// TIA Portal V20 export
FUNCTION_BLOCK "FB_ShredderSequencer"   // FB8, LAD
TITLE = Shredder Plant Sequencer
// Shredder plant sequencer (C-118-C-125): commands the shredder motor (via FB_MotorFwdRevSystem, wired at FC_ControlMain) and gates infeed/discharge conveyors and upstream enable, through a stepped cycle. Step legend (C-120): 0=Idle (stopped, waiting for a start condition) - 10=PreStart (siren warning before motion; arms the motor via MotorStartArm) - 20=DischargeStart (discharge conveyor starting, timed) - 30=ReverseRun (reverse commanded; the motor FB's own ReverseDelay entry pause elapses inside this step, then ReverseRunTimer counts ShredderReverseRunTime of CONFIRMED reverse feedback) - 40=WaitForwardRun (waiting for forward-run feedback) - 50=Running (normal production; infeed/upstream-enable timers and overcurrent detection are live) - 60=OvercurrentAbort (tripped - pause, then retry into ReverseRun, or stay out if too many reversals). Stop-all (REQ-012/013/062): StopCmd = stop button OR downstream lost OR control circuit unhealthy - aborts every step to Idle. Pusher handling is split (owner amendment 2026-07-16): stop button/unhealthy force pusher mode 0 (parks AND blocks jog), while any live stop reason - downstream loss included - raises PusherCycleInhibitCmd (no cycle launches or continues into a stopped plant, hand-jog stays available).
   VAR RETAIN
      IO { S7_SetPoint := 'True'} : "UDT_ShredderSequencerIO";   // Caller-visible interface (C-115) - FC_ControlMain writes CycleStart/CycleStop/feedback/tunables in, reads Run*/EnableUpstream/PreStartSounder/motor-command bits out. See the block header for the Step value legend.
   END_VAR
   VAR
      StopCmd : Bool;   // Stop-all: operator CycleStop, loss of DownstreamRunning (nowhere for shredded material to go), or loss of SystemHealthy (control circuit/E-stop - REQ-062: recovery must demand a fresh start press, so the sequence may not sit in a run step through an E-stop). Read by every step's own stop transition below and mirrored to the pusher as PusherCycleInhibitCmd.
      PusherModeForceOff : Bool;   // Named once (C-601): the hard pusher force - operator stop or circuit-unhealthy, plus the overcurrent-abort step. Forces PusherModeCmd to 0, which parks the pusher AND blocks jogging. Deliberately NOT the full StopCmd (owner amendment 2026-07-16): downstream absence must leave hand-jog available (REQ-040), so it reaches the pusher only as PusherCycleInhibitCmd.
      ReversalWindowTimeMS : DInt;
      PreStartSounderTimeMS : DInt;
      DischargeConveyorTimeoutMS : DInt;
      ShredderReverseRunTimeMS : DInt;
      InfeedRestartDelayMS : DInt;
      InfeedToUpstreamEnableDelayMS : DInt;
      OvercurrentSpinUpAllowanceMS : DInt;
      OvercurrentMediumDelayMS : DInt;
      OvercurrentHighDelayMS : DInt;
      ReversalRetryPauseTimeMS : DInt;
      ReversalWindowTimer { S7_SetPoint := 'True'} : TON_TIME;
      ReversalStepEdge : Bool;
      ReversalStepEdgeMem : Bool;
      ReversalCount : Int;   // Reversals since the window last re-armed (not per-cycle, unlike the pusher's own PressureTripCount) - ReversalWindowTimer restarts the window every time this is above zero, so ReversalCountThreshold reversals must occur within one ReversalWindowTime of each other to raise ShredderBlockedFault, not just ReversalCountThreshold times ever.
      PreStartTimer { S7_SetPoint := 'True'} : TON_TIME;
      DischargeStartTimer { S7_SetPoint := 'True'} : TON_TIME;
      ReverseRunTimer { S7_SetPoint := 'True'} : TON_TIME;
      InfeedRestartTimer { S7_SetPoint := 'True'} : TON_TIME;
      UpstreamEnableTimer { S7_SetPoint := 'True'} : TON_TIME;
      InfeedRunning : Bool;   // Latched once InfeedRestartTimer has timed out from the last hopper-clear - drives RunInfeedConv directly and (after a further UpstreamEnableTimer delay) EnableUpstream.
      SpinUpTimer { S7_SetPoint := 'True'} : TON_TIME;
      OvercurrentMediumTimer { S7_SetPoint := 'True'} : TON_TIME;
      OvercurrentHighTimer { S7_SetPoint := 'True'} : TON_TIME;
      OvercurrentTripped : Bool;   // KNOWN GAP, not wired to real current yet: both timers below are gated 'AND NOT AlwaysTrue' (permanently false placeholders) because DB_AnalogInput.ShredderMotorCurrent > DB_Settings.OvercurrentSetpointMedium/High is a genuine Real-vs-Real comparison this converter's synthesizer can't type correctly yet (hardcodes Int) - flagged and deferred rather than guessed at. This bit, and Step 50's own overcurrent-abort transition, are dead code until that's built.
      OvercurrentAbortPauseTimer { S7_SetPoint := 'True'} : TON_TIME;
   END_VAR
   VAR_TEMP
      "Time" : Real;
   END_VAR
BEGIN

REGION Network 1: Stop Command
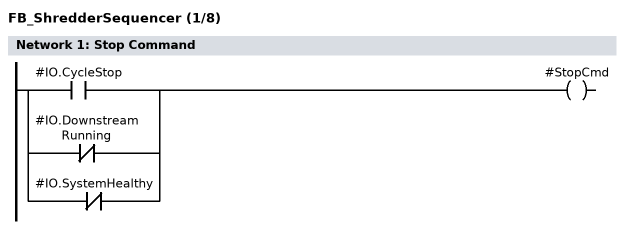
   RUNG wire#powerrail
      Contact( #IO.CycleStop )
      wire#w1
      Coil( #StopCmd )
   END_RUNG
   RUNG wire#powerrail
      I_Contact( #IO.DownstreamRunning )
   END_RUNG wire#w1
   RUNG wire#powerrail
      I_Contact( #IO.SystemHealthy )
   END_RUNG wire#w1
   // the same network as SCL:
   #StopCmd := #IO.CycleStop OR NOT #IO.DownstreamRunning OR NOT #IO.SystemHealthy;
END_REGION

REGION Network 2: HMI Time Conversions
   // HMI/DB_Settings times are Real seconds for operator legibility; every TON below needs its PT in DInt ms - one MUL+CONVERT pair per timer, matching the MotorDOL FTTime/EnableUPSTime idiom. Kept as one block up front rather than repeated at each timer, so the x1000 idiom is visibly consistent and only ever done once.
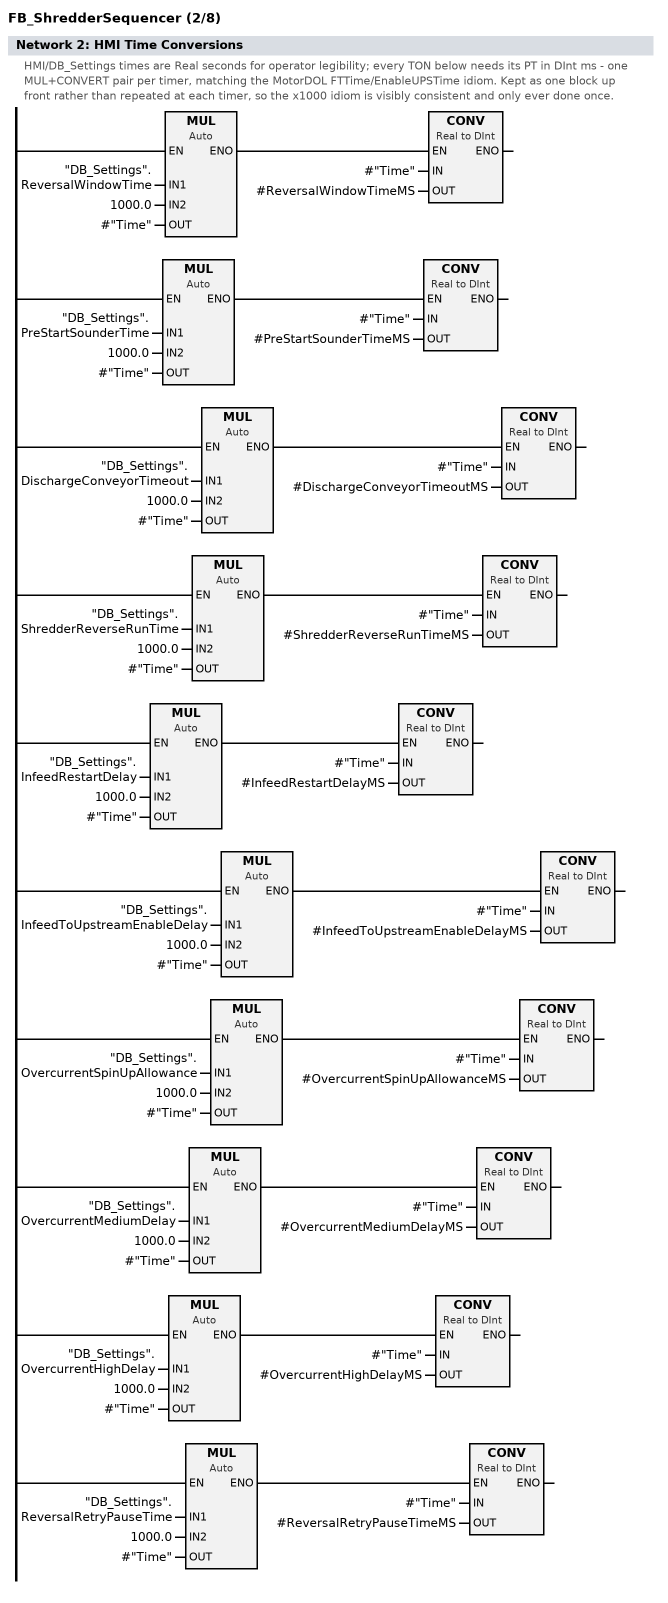
   RUNG wire#powerrail
      Mul(in1 := "DB_Settings".ReversalWindowTime, in2 := 1000.0, out := #"Time")
      { S7_Templates := "[SrcType := Real, DestType := DInt]" } Convert(in := #"Time", out := #ReversalWindowTimeMS)
   END_RUNG
   RUNG wire#powerrail
      Mul(in1 := "DB_Settings".PreStartSounderTime, in2 := 1000.0, out := #"Time")
      { S7_Templates := "[SrcType := Real, DestType := DInt]" } Convert(in := #"Time", out := #PreStartSounderTimeMS)
   END_RUNG
   RUNG wire#powerrail
      Mul(in1 := "DB_Settings".DischargeConveyorTimeout, in2 := 1000.0, out := #"Time")
      { S7_Templates := "[SrcType := Real, DestType := DInt]" } Convert(in := #"Time", out := #DischargeConveyorTimeoutMS)
   END_RUNG
   RUNG wire#powerrail
      Mul(in1 := "DB_Settings".ShredderReverseRunTime, in2 := 1000.0, out := #"Time")
      { S7_Templates := "[SrcType := Real, DestType := DInt]" } Convert(in := #"Time", out := #ShredderReverseRunTimeMS)
   END_RUNG
   RUNG wire#powerrail
      Mul(in1 := "DB_Settings".InfeedRestartDelay, in2 := 1000.0, out := #"Time")
      { S7_Templates := "[SrcType := Real, DestType := DInt]" } Convert(in := #"Time", out := #InfeedRestartDelayMS)
   END_RUNG
   RUNG wire#powerrail
      Mul(in1 := "DB_Settings".InfeedToUpstreamEnableDelay, in2 := 1000.0, out := #"Time")
      { S7_Templates := "[SrcType := Real, DestType := DInt]" } Convert(in := #"Time", out := #InfeedToUpstreamEnableDelayMS)
   END_RUNG
   RUNG wire#powerrail
      Mul(in1 := "DB_Settings".OvercurrentSpinUpAllowance, in2 := 1000.0, out := #"Time")
      { S7_Templates := "[SrcType := Real, DestType := DInt]" } Convert(in := #"Time", out := #OvercurrentSpinUpAllowanceMS)
   END_RUNG
   RUNG wire#powerrail
      Mul(in1 := "DB_Settings".OvercurrentMediumDelay, in2 := 1000.0, out := #"Time")
      { S7_Templates := "[SrcType := Real, DestType := DInt]" } Convert(in := #"Time", out := #OvercurrentMediumDelayMS)
   END_RUNG
   RUNG wire#powerrail
      Mul(in1 := "DB_Settings".OvercurrentHighDelay, in2 := 1000.0, out := #"Time")
      { S7_Templates := "[SrcType := Real, DestType := DInt]" } Convert(in := #"Time", out := #OvercurrentHighDelayMS)
   END_RUNG
   RUNG wire#powerrail
      Mul(in1 := "DB_Settings".ReversalRetryPauseTime, in2 := 1000.0, out := #"Time")
      { S7_Templates := "[SrcType := Real, DestType := DInt]" } Convert(in := #"Time", out := #ReversalRetryPauseTimeMS)
   END_RUNG
   // the same network as SCL:
   <??.?> := "DB_Settings".ReversalWindowTime * 1000.0 * #"Time";
   <??.?> := REAL_TO_DINT(#"Time");
   <??.?> := "DB_Settings".PreStartSounderTime * 1000.0 * #"Time";
   <??.?> := REAL_TO_DINT(#"Time");
   <??.?> := "DB_Settings".DischargeConveyorTimeout * 1000.0 * #"Time";
   <??.?> := REAL_TO_DINT(#"Time");
   <??.?> := "DB_Settings".ShredderReverseRunTime * 1000.0 * #"Time";
   <??.?> := REAL_TO_DINT(#"Time");
   <??.?> := "DB_Settings".InfeedRestartDelay * 1000.0 * #"Time";
   <??.?> := REAL_TO_DINT(#"Time");
   <??.?> := "DB_Settings".InfeedToUpstreamEnableDelay * 1000.0 * #"Time";
   <??.?> := REAL_TO_DINT(#"Time");
   <??.?> := "DB_Settings".OvercurrentSpinUpAllowance * 1000.0 * #"Time";
   <??.?> := REAL_TO_DINT(#"Time");
   <??.?> := "DB_Settings".OvercurrentMediumDelay * 1000.0 * #"Time";
   <??.?> := REAL_TO_DINT(#"Time");
   <??.?> := "DB_Settings".OvercurrentHighDelay * 1000.0 * #"Time";
   <??.?> := REAL_TO_DINT(#"Time");
   <??.?> := "DB_Settings".ReversalRetryPauseTime * 1000.0 * #"Time";
   <??.?> := REAL_TO_DINT(#"Time");
END_REGION

REGION Network 3: Reversal Re-Arm Window Timer
   // Retriggerable on-delay built from TON+edge (C-406/C-404 - no TONR/TOF exists to do this natively). IN drops false the instant a NEW reversal is detected - Step transitioning into 60, tested against ReversalStepEdgeMem's own previous-scan value (correct read-before-write ordering: this network reads the memory bit before Network 4 updates it later the same scan, so no cross-network staleness) - which resets ET/Q to 0 that scan; the timer then re-arms and must run a full ReversalWindowTime with no further reversal before Q goes true. Fixed 2026-07-17 (owner ruling, B-5/REQ-028): the prior rung read IN := ReversalCount > 0 alone, a level condition that only ever ran once from the first reversal - a fixed window, not the re-arming one this network's own title always claimed (C-608).
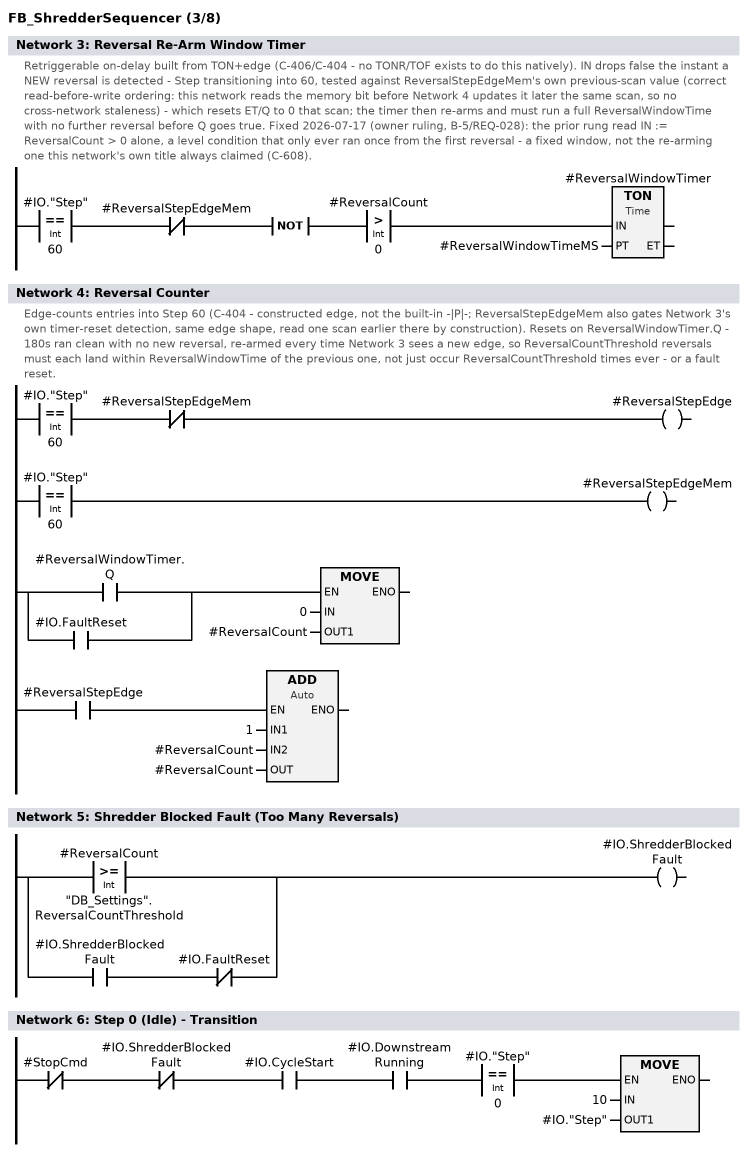
   RUNG wire#powerrail
      { S7_Templates := "SrcType := Int" } EQ_Contact(in1 := #IO."Step", in2 := 60)
      I_Contact( #ReversalStepEdgeMem )
      Not()
      { S7_Templates := "SrcType := Int" } GT_Contact(in1 := #ReversalCount, in2 := 0)
      { S7_Templates := "time_type := Time" } #ReversalWindowTimer.TON(pt := #ReversalWindowTimeMS, et =>)
   END_RUNG
   // the same network as SCL:
   #ReversalWindowTimer(IN := NOT ((#IO."Step" = 60) AND NOT #ReversalStepEdgeMem) AND (#ReversalCount > 0),   // TON
                        PT := #ReversalWindowTimeMS);
END_REGION

REGION Network 4: Reversal Counter
   // Edge-counts entries into Step 60 (C-404 - constructed edge, not the built-in -|P|-; ReversalStepEdgeMem also gates Network 3's own timer-reset detection, same edge shape, read one scan earlier there by construction). Resets on ReversalWindowTimer.Q - 180s ran clean with no new reversal, re-armed every time Network 3 sees a new edge, so ReversalCountThreshold reversals must each land within ReversalWindowTime of the previous one, not just occur ReversalCountThreshold times ever - or a fault reset.
   RUNG wire#powerrail
      { S7_Templates := "SrcType := Int" } EQ_Contact(in1 := #IO."Step", in2 := 60)
      I_Contact( #ReversalStepEdgeMem )
      Coil( #ReversalStepEdge )
   END_RUNG
   RUNG wire#powerrail
      { S7_Templates := "SrcType := Int" } EQ_Contact(in1 := #IO."Step", in2 := 60)
      Coil( #ReversalStepEdgeMem )
   END_RUNG
   RUNG wire#powerrail
      Contact( #ReversalWindowTimer.Q )
      wire#w1
      Move(in := 0, out1 := #ReversalCount)
   END_RUNG
   RUNG wire#powerrail
      Contact( #IO.FaultReset )
   END_RUNG wire#w1
   RUNG wire#powerrail
      Contact( #ReversalStepEdge )
      Add(in1 := 1, in2 := #ReversalCount, out := #ReversalCount)
   END_RUNG
   // the same network as SCL:
   #ReversalStepEdge := (#IO."Step" = 60) AND NOT #ReversalStepEdgeMem;
   #ReversalStepEdgeMem := #IO."Step" = 60;
   IF #ReversalWindowTimer.Q OR #IO.FaultReset THEN <??.?> := 0; END_IF;
   IF #ReversalStepEdge THEN <??.?> := 1 + #ReversalCount + #ReversalCount; END_IF;
END_REGION

REGION Network 5: Shredder Blocked Fault (Too Many Reversals)
   RUNG wire#powerrail
      { S7_Templates := "SrcType := Int" } GE_Contact(in1 := #ReversalCount, in2 := "DB_Settings".ReversalCountThreshold)
      wire#w1
      Coil( #IO.ShredderBlockedFault )
   END_RUNG
   RUNG wire#powerrail
      Contact( #IO.ShredderBlockedFault )
      I_Contact( #IO.FaultReset )
   END_RUNG wire#w1
   // the same network as SCL:
   #IO.ShredderBlockedFault := (#ReversalCount >= "DB_Settings".ReversalCountThreshold) OR (#IO.ShredderBlockedFault AND NOT #IO.FaultReset);
END_REGION

REGION Network 6: Step 0 (Idle) - Transition
   RUNG wire#powerrail
      I_Contact( #StopCmd )
      I_Contact( #IO.ShredderBlockedFault )
      Contact( #IO.CycleStart )
      Contact( #IO.DownstreamRunning )
      { S7_Templates := "SrcType := Int" } EQ_Contact(in1 := #IO."Step", in2 := 0)
      Move(in := 10, out1 := #IO."Step")
   END_RUNG
   // the same network as SCL:
   IF NOT #StopCmd AND NOT #IO.ShredderBlockedFault AND #IO.CycleStart AND #IO.DownstreamRunning AND (#IO."Step" = 0) THEN
       <??.?> := 10;
   END_IF;
END_REGION

REGION Network 7: Step 10 (PreStart) - Timer And Transitions
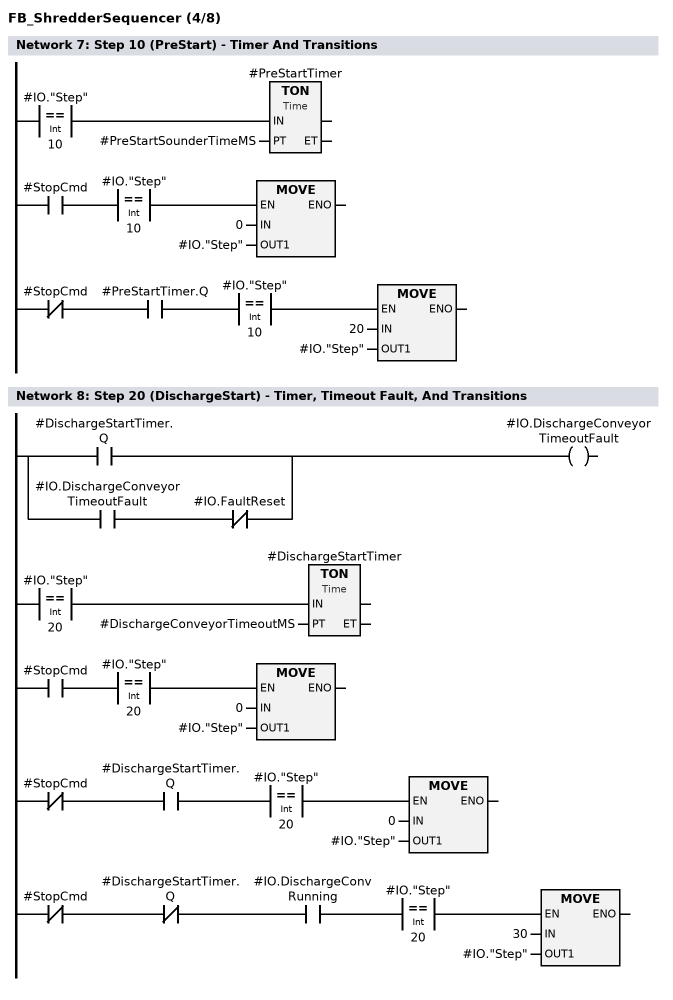
   RUNG wire#powerrail
      { S7_Templates := "SrcType := Int" } EQ_Contact(in1 := #IO."Step", in2 := 10)
      { S7_Templates := "time_type := Time" } #PreStartTimer.TON(pt := #PreStartSounderTimeMS, et =>)
   END_RUNG
   RUNG wire#powerrail
      Contact( #StopCmd )
      { S7_Templates := "SrcType := Int" } EQ_Contact(in1 := #IO."Step", in2 := 10)
      Move(in := 0, out1 := #IO."Step")
   END_RUNG
   RUNG wire#powerrail
      I_Contact( #StopCmd )
      Contact( #PreStartTimer.Q )
      { S7_Templates := "SrcType := Int" } EQ_Contact(in1 := #IO."Step", in2 := 10)
      Move(in := 20, out1 := #IO."Step")
   END_RUNG
   // the same network as SCL:
   #PreStartTimer(IN := #IO."Step" = 10, PT := #PreStartSounderTimeMS);   // TON
   IF #StopCmd AND (#IO."Step" = 10) THEN <??.?> := 0; END_IF;
   IF NOT #StopCmd AND #PreStartTimer.Q AND (#IO."Step" = 10) THEN <??.?> := 20; END_IF;
END_REGION

REGION Network 8: Step 20 (DischargeStart) - Timer, Timeout Fault, And Transitions
   RUNG wire#powerrail
      Contact( #DischargeStartTimer.Q )
      wire#w1
      Coil( #IO.DischargeConveyorTimeoutFault )
   END_RUNG
   RUNG wire#powerrail
      Contact( #IO.DischargeConveyorTimeoutFault )
      I_Contact( #IO.FaultReset )
   END_RUNG wire#w1
   RUNG wire#powerrail
      { S7_Templates := "SrcType := Int" } EQ_Contact(in1 := #IO."Step", in2 := 20)
      { S7_Templates := "time_type := Time" } #DischargeStartTimer.TON(pt := #DischargeConveyorTimeoutMS, et =>)
   END_RUNG
   RUNG wire#powerrail
      Contact( #StopCmd )
      { S7_Templates := "SrcType := Int" } EQ_Contact(in1 := #IO."Step", in2 := 20)
      Move(in := 0, out1 := #IO."Step")
   END_RUNG
   RUNG wire#powerrail
      I_Contact( #StopCmd )
      Contact( #DischargeStartTimer.Q )
      { S7_Templates := "SrcType := Int" } EQ_Contact(in1 := #IO."Step", in2 := 20)
      Move(in := 0, out1 := #IO."Step")
   END_RUNG
   RUNG wire#powerrail
      I_Contact( #StopCmd )
      I_Contact( #DischargeStartTimer.Q )
      Contact( #IO.DischargeConvRunning )
      { S7_Templates := "SrcType := Int" } EQ_Contact(in1 := #IO."Step", in2 := 20)
      Move(in := 30, out1 := #IO."Step")
   END_RUNG
   // the same network as SCL:
   #IO.DischargeConveyorTimeoutFault := #DischargeStartTimer.Q OR (#IO.DischargeConveyorTimeoutFault AND NOT #IO.FaultReset);
   #DischargeStartTimer(IN := #IO."Step" = 20, PT := #DischargeConveyorTimeoutMS);   // TON
   IF #StopCmd AND (#IO."Step" = 20) THEN <??.?> := 0; END_IF;
   IF NOT #StopCmd AND #DischargeStartTimer.Q AND (#IO."Step" = 20) THEN <??.?> := 0; END_IF;
   IF NOT #StopCmd AND NOT #DischargeStartTimer.Q AND #IO.DischargeConvRunning AND (#IO."Step" = 20) THEN
       <??.?> := 30;
   END_IF;
END_REGION

REGION Network 9: Step 30 (ReverseRun) - Timer And Transitions
   // ReverseRunTimer counts only while reverse is CONFIRMED running (ShredderRunRevFB), so the spec's 6 s (REQ-005) buys 6 s of actual rotation - the motor FB's 8 s ReverseDelay entry pause no longer eats the window, and a feedback dropout restarts the count. The commanded-but-no-feedback dwell is deliberately NOT re-timed here (C-409, one interval one place; step 40 already relies on the same mechanism): the motor FB's own fail-to-run window (FTTime, after its ReverseIgnoreFT masking) latches FTR, and the MotorFaultActive exit below aborts the step - bounded dwell, latched fault, C-122's substance without a duplicate timer.
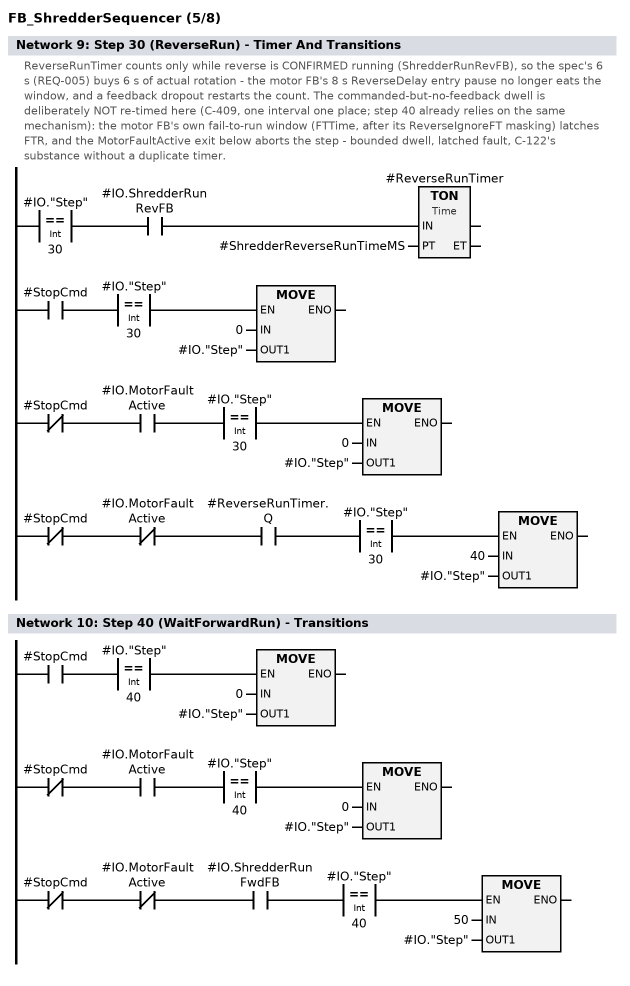
   RUNG wire#powerrail
      { S7_Templates := "SrcType := Int" } EQ_Contact(in1 := #IO."Step", in2 := 30)
      Contact( #IO.ShredderRunRevFB )
      { S7_Templates := "time_type := Time" } #ReverseRunTimer.TON(pt := #ShredderReverseRunTimeMS, et =>)
   END_RUNG
   RUNG wire#powerrail
      Contact( #StopCmd )
      { S7_Templates := "SrcType := Int" } EQ_Contact(in1 := #IO."Step", in2 := 30)
      Move(in := 0, out1 := #IO."Step")
   END_RUNG
   RUNG wire#powerrail
      I_Contact( #StopCmd )
      Contact( #IO.MotorFaultActive )
      { S7_Templates := "SrcType := Int" } EQ_Contact(in1 := #IO."Step", in2 := 30)
      Move(in := 0, out1 := #IO."Step")
   END_RUNG
   RUNG wire#powerrail
      I_Contact( #StopCmd )
      I_Contact( #IO.MotorFaultActive )
      Contact( #ReverseRunTimer.Q )
      { S7_Templates := "SrcType := Int" } EQ_Contact(in1 := #IO."Step", in2 := 30)
      Move(in := 40, out1 := #IO."Step")
   END_RUNG
   // the same network as SCL:
   #ReverseRunTimer(IN := (#IO."Step" = 30) AND #IO.ShredderRunRevFB, PT := #ShredderReverseRunTimeMS);   // TON
   IF #StopCmd AND (#IO."Step" = 30) THEN <??.?> := 0; END_IF;
   IF NOT #StopCmd AND #IO.MotorFaultActive AND (#IO."Step" = 30) THEN <??.?> := 0; END_IF;
   IF NOT #StopCmd AND NOT #IO.MotorFaultActive AND #ReverseRunTimer.Q AND (#IO."Step" = 30) THEN
       <??.?> := 40;
   END_IF;
END_REGION

REGION Network 10: Step 40 (WaitForwardRun) - Transitions
   RUNG wire#powerrail
      Contact( #StopCmd )
      { S7_Templates := "SrcType := Int" } EQ_Contact(in1 := #IO."Step", in2 := 40)
      Move(in := 0, out1 := #IO."Step")
   END_RUNG
   RUNG wire#powerrail
      I_Contact( #StopCmd )
      Contact( #IO.MotorFaultActive )
      { S7_Templates := "SrcType := Int" } EQ_Contact(in1 := #IO."Step", in2 := 40)
      Move(in := 0, out1 := #IO."Step")
   END_RUNG
   RUNG wire#powerrail
      I_Contact( #StopCmd )
      I_Contact( #IO.MotorFaultActive )
      Contact( #IO.ShredderRunFwdFB )
      { S7_Templates := "SrcType := Int" } EQ_Contact(in1 := #IO."Step", in2 := 40)
      Move(in := 50, out1 := #IO."Step")
   END_RUNG
   // the same network as SCL:
   IF #StopCmd AND (#IO."Step" = 40) THEN <??.?> := 0; END_IF;
   IF NOT #StopCmd AND #IO.MotorFaultActive AND (#IO."Step" = 40) THEN <??.?> := 0; END_IF;
   IF NOT #StopCmd AND NOT #IO.MotorFaultActive AND #IO.ShredderRunFwdFB AND (#IO."Step" = 40) THEN
       <??.?> := 50;
   END_IF;
END_REGION

REGION Network 11: Step 50 (Running) - Infeed Restart, Upstream Enable, And Outputs
   // UpstreamEnableTimer's own IN reads InfeedRunning one scan behind this network's own InfeedRunning update below (it's kind-ordered before the coil that writes it) - harmless for a multi-second delay, and matches this design's original timing exactly. EnableUpstream lives here, next to its own timer, rather than in the general Output Commands network - this is the output the MotorFwdRevSystem CALL-site correction was specifically about: it must only ever come from Step=50 dwell time, never from motor-running telemetry.
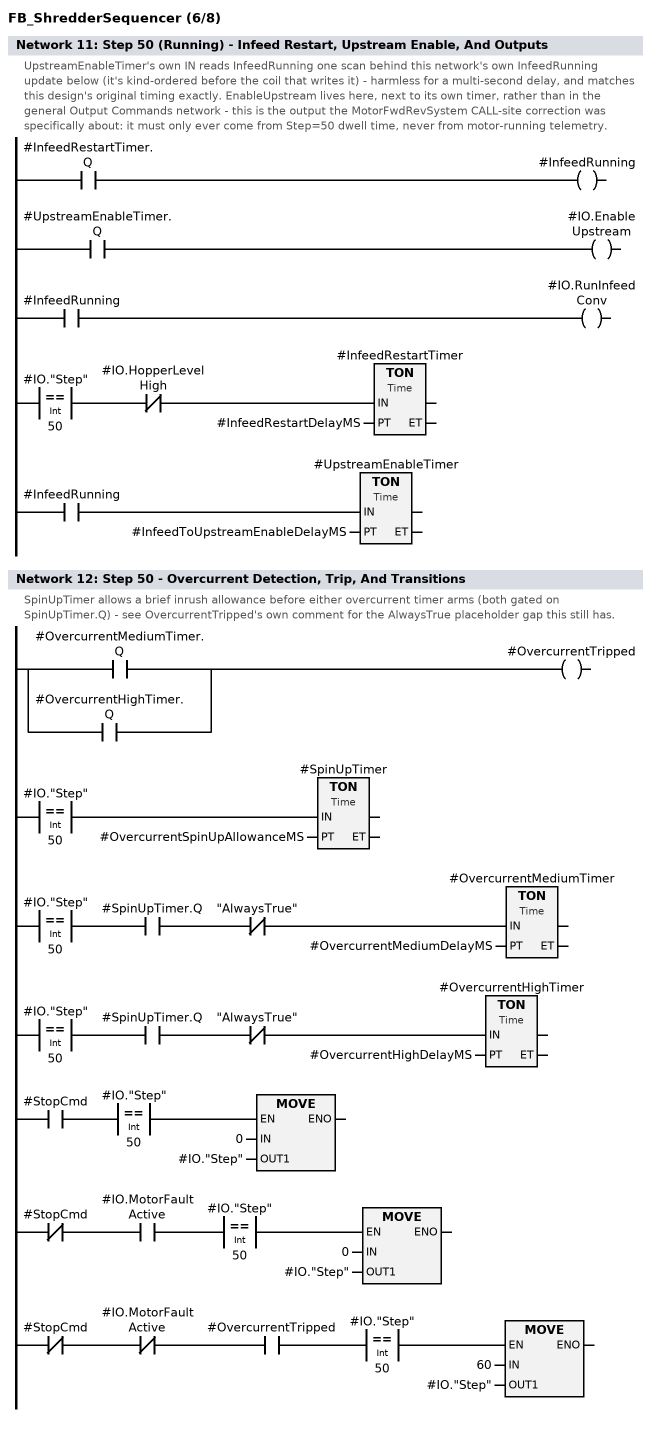
   RUNG wire#powerrail
      Contact( #InfeedRestartTimer.Q )
      Coil( #InfeedRunning )
   END_RUNG
   RUNG wire#powerrail
      Contact( #UpstreamEnableTimer.Q )
      Coil( #IO.EnableUpstream )
   END_RUNG
   RUNG wire#powerrail
      Contact( #InfeedRunning )
      Coil( #IO.RunInfeedConv )
   END_RUNG
   RUNG wire#powerrail
      { S7_Templates := "SrcType := Int" } EQ_Contact(in1 := #IO."Step", in2 := 50)
      I_Contact( #IO.HopperLevelHigh )
      { S7_Templates := "time_type := Time" } #InfeedRestartTimer.TON(pt := #InfeedRestartDelayMS, et =>)
   END_RUNG
   RUNG wire#powerrail
      Contact( #InfeedRunning )
      { S7_Templates := "time_type := Time" } #UpstreamEnableTimer.TON(pt := #InfeedToUpstreamEnableDelayMS, et =>)
   END_RUNG
   // the same network as SCL:
   #InfeedRunning := #InfeedRestartTimer.Q;
   #IO.EnableUpstream := #UpstreamEnableTimer.Q;
   #IO.RunInfeedConv := #InfeedRunning;
   #InfeedRestartTimer(IN := (#IO."Step" = 50) AND NOT #IO.HopperLevelHigh, PT := #InfeedRestartDelayMS);   // TON
   #UpstreamEnableTimer(IN := #InfeedRunning, PT := #InfeedToUpstreamEnableDelayMS);   // TON
END_REGION

REGION Network 12: Step 50 - Overcurrent Detection, Trip, And Transitions
   // SpinUpTimer allows a brief inrush allowance before either overcurrent timer arms (both gated on SpinUpTimer.Q) - see OvercurrentTripped's own comment for the AlwaysTrue placeholder gap this still has.
   RUNG wire#powerrail
      Contact( #OvercurrentMediumTimer.Q )
      wire#w1
      Coil( #OvercurrentTripped )
   END_RUNG
   RUNG wire#powerrail
      Contact( #OvercurrentHighTimer.Q )
   END_RUNG wire#w1
   RUNG wire#powerrail
      { S7_Templates := "SrcType := Int" } EQ_Contact(in1 := #IO."Step", in2 := 50)
      { S7_Templates := "time_type := Time" } #SpinUpTimer.TON(pt := #OvercurrentSpinUpAllowanceMS, et =>)
   END_RUNG
   RUNG wire#powerrail
      { S7_Templates := "SrcType := Int" } EQ_Contact(in1 := #IO."Step", in2 := 50)
      Contact( #SpinUpTimer.Q )
      I_Contact( "AlwaysTrue" )
      { S7_Templates := "time_type := Time" } #OvercurrentMediumTimer.TON(pt := #OvercurrentMediumDelayMS, et =>)
   END_RUNG
   RUNG wire#powerrail
      { S7_Templates := "SrcType := Int" } EQ_Contact(in1 := #IO."Step", in2 := 50)
      Contact( #SpinUpTimer.Q )
      I_Contact( "AlwaysTrue" )
      { S7_Templates := "time_type := Time" } #OvercurrentHighTimer.TON(pt := #OvercurrentHighDelayMS, et =>)
   END_RUNG
   RUNG wire#powerrail
      Contact( #StopCmd )
      { S7_Templates := "SrcType := Int" } EQ_Contact(in1 := #IO."Step", in2 := 50)
      Move(in := 0, out1 := #IO."Step")
   END_RUNG
   RUNG wire#powerrail
      I_Contact( #StopCmd )
      Contact( #IO.MotorFaultActive )
      { S7_Templates := "SrcType := Int" } EQ_Contact(in1 := #IO."Step", in2 := 50)
      Move(in := 0, out1 := #IO."Step")
   END_RUNG
   RUNG wire#powerrail
      I_Contact( #StopCmd )
      I_Contact( #IO.MotorFaultActive )
      Contact( #OvercurrentTripped )
      { S7_Templates := "SrcType := Int" } EQ_Contact(in1 := #IO."Step", in2 := 50)
      Move(in := 60, out1 := #IO."Step")
   END_RUNG
   // the same network as SCL:
   #OvercurrentTripped := #OvercurrentMediumTimer.Q OR #OvercurrentHighTimer.Q;
   #SpinUpTimer(IN := #IO."Step" = 50, PT := #OvercurrentSpinUpAllowanceMS);   // TON
   #OvercurrentMediumTimer(IN := (#IO."Step" = 50) AND #SpinUpTimer.Q AND NOT "AlwaysTrue",   // TON
                           PT := #OvercurrentMediumDelayMS);
   #OvercurrentHighTimer(IN := (#IO."Step" = 50) AND #SpinUpTimer.Q AND NOT "AlwaysTrue",   // TON
                         PT := #OvercurrentHighDelayMS);
   IF #StopCmd AND (#IO."Step" = 50) THEN <??.?> := 0; END_IF;
   IF NOT #StopCmd AND #IO.MotorFaultActive AND (#IO."Step" = 50) THEN <??.?> := 0; END_IF;
   IF NOT #StopCmd AND NOT #IO.MotorFaultActive AND #OvercurrentTripped AND (#IO."Step" = 50) THEN
       <??.?> := 60;
   END_IF;
END_REGION

REGION Network 13: Step 60 (OvercurrentAbort) - Timer And Transitions
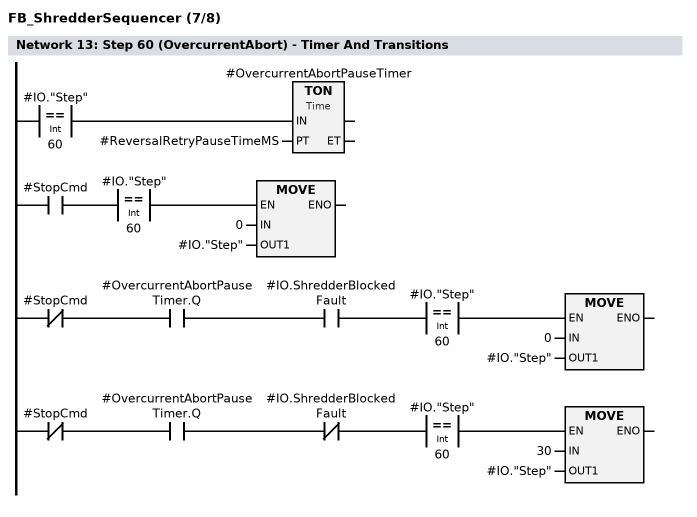
   RUNG wire#powerrail
      { S7_Templates := "SrcType := Int" } EQ_Contact(in1 := #IO."Step", in2 := 60)
      { S7_Templates := "time_type := Time" } #OvercurrentAbortPauseTimer.TON(pt := #ReversalRetryPauseTimeMS, et =>)
   END_RUNG
   RUNG wire#powerrail
      Contact( #StopCmd )
      { S7_Templates := "SrcType := Int" } EQ_Contact(in1 := #IO."Step", in2 := 60)
      Move(in := 0, out1 := #IO."Step")
   END_RUNG
   RUNG wire#powerrail
      I_Contact( #StopCmd )
      Contact( #OvercurrentAbortPauseTimer.Q )
      Contact( #IO.ShredderBlockedFault )
      { S7_Templates := "SrcType := Int" } EQ_Contact(in1 := #IO."Step", in2 := 60)
      Move(in := 0, out1 := #IO."Step")
   END_RUNG
   RUNG wire#powerrail
      I_Contact( #StopCmd )
      Contact( #OvercurrentAbortPauseTimer.Q )
      I_Contact( #IO.ShredderBlockedFault )
      { S7_Templates := "SrcType := Int" } EQ_Contact(in1 := #IO."Step", in2 := 60)
      Move(in := 30, out1 := #IO."Step")
   END_RUNG
   // the same network as SCL:
   #OvercurrentAbortPauseTimer(IN := #IO."Step" = 60, PT := #ReversalRetryPauseTimeMS);   // TON
   IF #StopCmd AND (#IO."Step" = 60) THEN <??.?> := 0; END_IF;
   IF NOT #StopCmd AND #OvercurrentAbortPauseTimer.Q AND #IO.ShredderBlockedFault AND (#IO."Step" = 60) THEN
       <??.?> := 0;
   END_IF;
   IF NOT #StopCmd AND #OvercurrentAbortPauseTimer.Q AND NOT #IO.ShredderBlockedFault AND (#IO."Step" = 60) THEN
       <??.?> := 30;
   END_IF;
END_REGION

REGION Network 14: Motor And Pusher Mode Commands
   // MotorStartArm asserts only through PreStart: one operator start press = one motor arming (FC_ControlMain hands it to the motor FB's self-clearing RecentStart - REQ-062). PusherParkCmd holds through the machine-start steps 20-40 (range intent, C-603: any step inserted inside the start ramp still wants the pusher home) - long enough for the pusher's warned repark to fire even when the discharge confirm is quick (REQ-045); from Running onward the pusher's own cycle-entry repark takes over. Pusher stop handling is two-tier (REQ-012/013 + owner amendment 2026-07-16): PusherModeForceOff (stop button/unhealthy/step-60, mirroring the step-60 overcurrent force) drives mode 0 - parks the pusher and blocks jog - while PusherCycleInhibitCmd mirrors the full StopCmd so downstream loss still stops cycle behavior without taking hand-jog away (REQ-040).
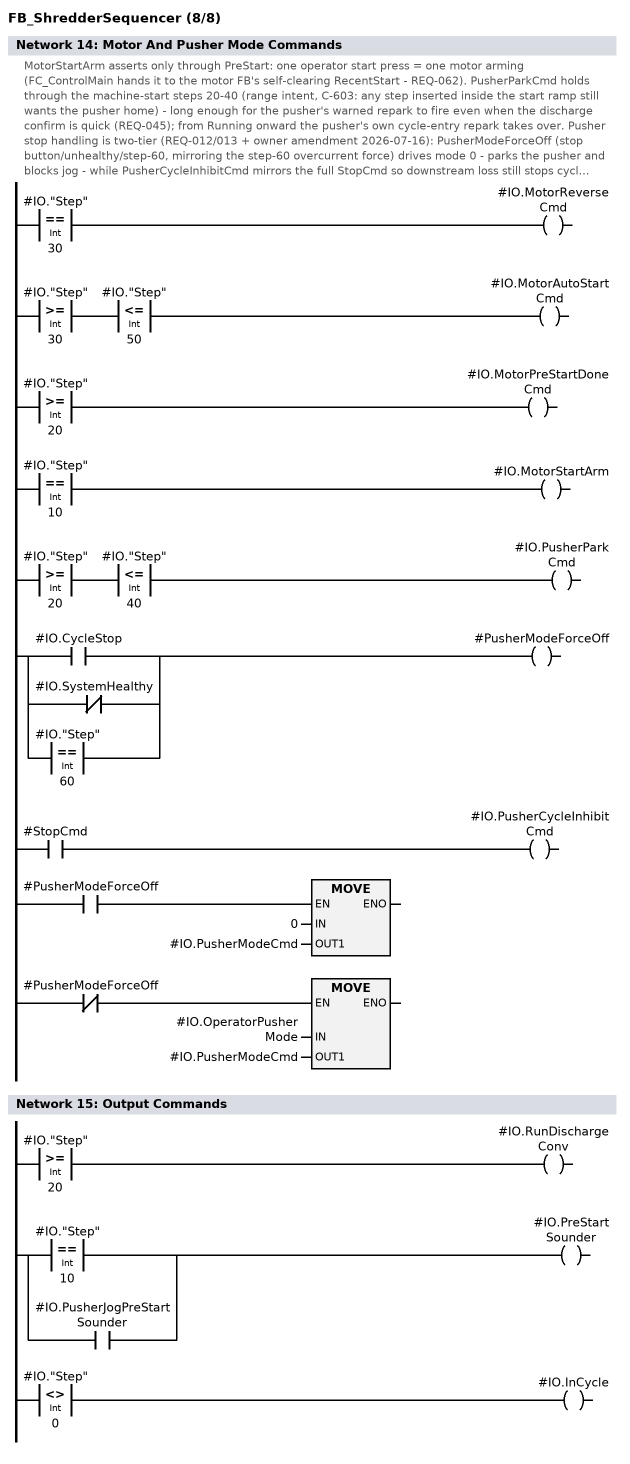
   RUNG wire#powerrail
      { S7_Templates := "SrcType := Int" } EQ_Contact(in1 := #IO."Step", in2 := 30)
      Coil( #IO.MotorReverseCmd )
   END_RUNG
   RUNG wire#powerrail
      { S7_Templates := "SrcType := Int" } GE_Contact(in1 := #IO."Step", in2 := 30)
      { S7_Templates := "SrcType := Int" } LE_Contact(in1 := #IO."Step", in2 := 50)
      Coil( #IO.MotorAutoStartCmd )
   END_RUNG
   RUNG wire#powerrail
      { S7_Templates := "SrcType := Int" } GE_Contact(in1 := #IO."Step", in2 := 20)
      Coil( #IO.MotorPreStartDoneCmd )
   END_RUNG
   RUNG wire#powerrail
      { S7_Templates := "SrcType := Int" } EQ_Contact(in1 := #IO."Step", in2 := 10)
      Coil( #IO.MotorStartArm )
   END_RUNG
   RUNG wire#powerrail
      { S7_Templates := "SrcType := Int" } GE_Contact(in1 := #IO."Step", in2 := 20)
      { S7_Templates := "SrcType := Int" } LE_Contact(in1 := #IO."Step", in2 := 40)
      Coil( #IO.PusherParkCmd )
   END_RUNG
   RUNG wire#powerrail
      Contact( #IO.CycleStop )
      wire#w1
      Coil( #PusherModeForceOff )
   END_RUNG
   RUNG wire#powerrail
      I_Contact( #IO.SystemHealthy )
   END_RUNG wire#w1
   RUNG wire#powerrail
      { S7_Templates := "SrcType := Int" } EQ_Contact(in1 := #IO."Step", in2 := 60)
   END_RUNG wire#w1
   RUNG wire#powerrail
      Contact( #StopCmd )
      Coil( #IO.PusherCycleInhibitCmd )
   END_RUNG
   RUNG wire#powerrail
      Contact( #PusherModeForceOff )
      Move(in := 0, out1 := #IO.PusherModeCmd)
   END_RUNG
   RUNG wire#powerrail
      I_Contact( #PusherModeForceOff )
      Move(in := #IO.OperatorPusherMode, out1 := #IO.PusherModeCmd)
   END_RUNG
   // the same network as SCL:
   #IO.MotorReverseCmd := #IO."Step" = 30;
   #IO.MotorAutoStartCmd := (#IO."Step" >= 30) AND (#IO."Step" <= 50);
   #IO.MotorPreStartDoneCmd := #IO."Step" >= 20;
   #IO.MotorStartArm := #IO."Step" = 10;
   #IO.PusherParkCmd := (#IO."Step" >= 20) AND (#IO."Step" <= 40);
   #PusherModeForceOff := #IO.CycleStop OR NOT #IO.SystemHealthy OR (#IO."Step" = 60);
   #IO.PusherCycleInhibitCmd := #StopCmd;
   IF #PusherModeForceOff THEN <??.?> := 0; END_IF;
   IF NOT #PusherModeForceOff THEN <??.?> := #IO.OperatorPusherMode; END_IF;
END_REGION

REGION Network 15: Output Commands
   RUNG wire#powerrail
      { S7_Templates := "SrcType := Int" } GE_Contact(in1 := #IO."Step", in2 := 20)
      Coil( #IO.RunDischargeConv )
   END_RUNG
   RUNG wire#powerrail
      { S7_Templates := "SrcType := Int" } EQ_Contact(in1 := #IO."Step", in2 := 10)
      wire#w1
      Coil( #IO.PreStartSounder )
   END_RUNG
   RUNG wire#powerrail
      Contact( #IO.PusherJogPreStartSounder )
   END_RUNG wire#w1
   RUNG wire#powerrail
      { S7_Templates := "SrcType := Int" } NE_Contact(in1 := #IO."Step", in2 := 0)
      Coil( #IO.InCycle )
   END_RUNG
   // the same network as SCL:
   #IO.RunDischargeConv := #IO."Step" >= 20;
   #IO.PreStartSounder := (#IO."Step" = 10) OR #IO.PusherJogPreStartSounder;
   #IO.InCycle := #IO."Step" <> 0;
END_REGION
END_FUNCTION_BLOCK
